(* Logix 5000 project; controller DispersionPlc vendor 1 type 14 code 108 rev 34.11; software revision 34.01; part 17 of 22 *)
(* tags used below, declared in another part *)
   _JISdebug : DINT;
   AFI : BOOL;
   AG4302_LLP_Alarm : BOOL;
   Current4302FQ : REAL;
   DPT_4302_Holding : REAL;
   Estop_Disp : ALIAS FOR Local:3:I.Data.1;
   FIT_4302_1 : AStd_AnalogInput;
   FIT_4305_xx : AStd_AnalogInput;
   K400_PhaseTransfer : AStd_PLI;
   LS_4302_High : BOOL;
   PIC_4302_3 : AStd_PIDInterface;
   RO_HE4305_PhaseROWaterAddition : AStd_PLI;
   SPARE_I402 : ALIAS FOR Local:4:I.Data.2;
   SPARE_I403 : ALIAS FOR Local:4:I.Data.3;
   SPARE_I408 : ALIAS FOR Local:4:I.Data.8;
   SPARE_I409 : ALIAS FOR Local:4:I.Data.9;
   SPARE_O512 : ALIAS FOR Local:5:O.Data.12;
   SPARE_O513 : ALIAS FOR Local:5:O.Data.13;
   SPARE_O605 : ALIAS FOR Local:6:O.Data.5;
   TIT_4305_1 : AStd_AnalogInput;
   V4306_PhaseTransfer : AStd_PLI;
   V4307_PhaseTransfer : AStd_PLI;
   VFD_4302_1 : AStd_VFD;
   VFD_P_4302_2 : AStd_VFD;
   WIT_4302_1 : AStd_AnalogInput;
   WIT_4302_1_AOI : AStd_AI_AOI;
   XV_4301_8 : AStd_VlvOC;
   XV_4302_10 : AStd_VlvOC;
   XV_4302_10_AOI : AStd_VlvOC_AOI;
   XV_4302_10_IOpn : BOOL;
   XV_4302_10_OCls : BOOL;
   XV_4302_12 : AStd_VlvOC;
   XV_4302_12_AOI : AStd_VlvOC_AOI;
   XV_4302_12_OCls : BOOL;
   XV_4302_13 : AStd_VlvOC;
   XV_4302_13_AOI : AStd_VlvOC_AOI;
   XV_4302_13_ClosedI : ALIAS FOR Local:1:I.Data[27].23;
   XV_4302_13_OCls : BOOL;
   XV_4302_13_OpenC : ALIAS FOR Local:1:O.Data[12].17;
   XV_4302_13_OpenI : ALIAS FOR Local:1:I.Data[27].24;
   XV_4302_2 : AStd_VlvOC;
   XV_4302_2_AOI : AStd_VlvOC_AOI;
   XV_4302_2_ICls : BOOL;
   XV_4302_2_IOpn : BOOL;
   XV_4302_2_OCls : BOOL;
   XV_4302_2_OOpn : BOOL;
   XV_4302_3 : AStd_VlvOC;
   XV_4302_3_AOI : AStd_VlvOC_AOI;
   XV_4302_3_ICls : BOOL;
   XV_4302_3_IOpn : BOOL;
   XV_4302_3_OCls : BOOL;
   XV_4302_3_OOpn : BOOL;
   XV_4302_4 : AStd_VlvOC;
   XV_4302_4_AOI : AStd_VlvOC_AOI;
   XV_4302_4_ICls : BOOL;
   XV_4302_4_IOpn : BOOL;
   XV_4302_4_OCls : BOOL;
   XV_4302_4_OOpn : BOOL;
   XV_4302_5 : AStd_VlvOC;
   XV_4302_5_AOI : AStd_VlvOC_AOI;
   XV_4302_5_IOpn : BOOL;
   XV_4302_5_OCls : BOOL;
   XV_4302_6 : AStd_VlvOC;
   XV_4302_6_AOI : AStd_VlvOC_AOI;
   XV_4302_6_IOpn : BOOL;
   XV_4302_6_OCls : BOOL;
   XV_4302_7 : AStd_VlvOC;
   XV_4302_7_AOI : AStd_VlvOC_AOI;
   XV_4302_7_IOpn : BOOL;
   XV_4302_7_OCls : BOOL;
   XV_4302_8 : AStd_VlvOC;
   XV_4302_8_AOI : AStd_VlvOC_AOI;
   XV_4302_8_IOpn : BOOL;
   XV_4302_8_OCls : BOOL;
   XV_4302_9 : AStd_VlvOC;
   XV_4306_3 : AStd_VlvOC;
   XV_4306_5 : AStd_VlvOC;
   XV_4307_3 : AStd_VlvOC;
   XV_4307_6 : AStd_VlvOC;
   XV_S52_2 : AStd_VlvOC;
(* Unit_T4302, continued *)

ROUTINE Device_WIT_4302_1   (* ladder *)
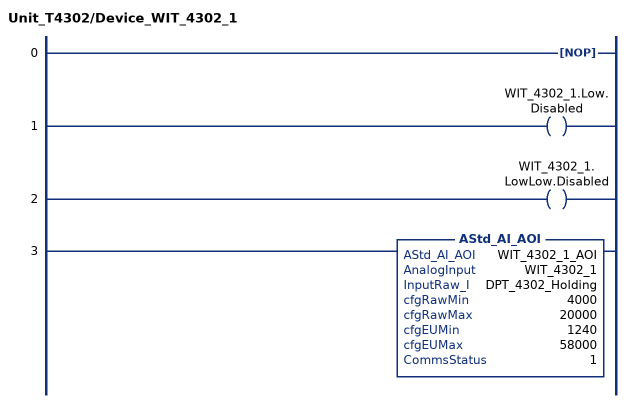
   0: NOP();
   1: OTE(WIT_4302_1.Low.Disabled);
   2: OTE(WIT_4302_1.LowLow.Disabled);
   3: AStd_AI_AOI(WIT_4302_1_AOI,WIT_4302_1,DPT_4302_Holding,4000,20000,1240,58000,1);
END_ROUTINE

ROUTINE Device_XV_4302_10   (* ladder *)
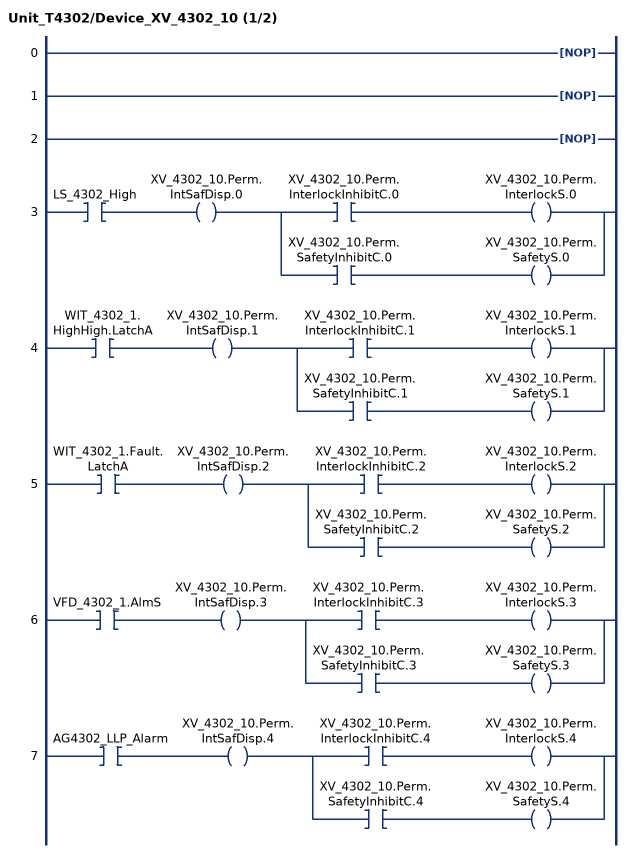
   0: NOP();
   1: NOP();
   2: NOP();
   3: XIC(LS_4302_High)OTE(XV_4302_10.Perm.IntSafDisp.0)[XIC(XV_4302_10.Perm.InterlockInhibitC.0) OTE(XV_4302_10.Perm.InterlockS.0) ,XIC(XV_4302_10.Perm.SafetyInhibitC.0) OTE(XV_4302_10.Perm.SafetyS.0) ];
   4: XIC(WIT_4302_1.HighHigh.LatchA)OTE(XV_4302_10.Perm.IntSafDisp.1)[XIC(XV_4302_10.Perm.InterlockInhibitC.1) OTE(XV_4302_10.Perm.InterlockS.1) ,XIC(XV_4302_10.Perm.SafetyInhibitC.1) OTE(XV_4302_10.Perm.SafetyS.1) ];
   5: XIC(WIT_4302_1.Fault.LatchA)OTE(XV_4302_10.Perm.IntSafDisp.2)[XIC(XV_4302_10.Perm.InterlockInhibitC.2) OTE(XV_4302_10.Perm.InterlockS.2) ,XIC(XV_4302_10.Perm.SafetyInhibitC.2) OTE(XV_4302_10.Perm.SafetyS.2) ];
   6: XIC(VFD_4302_1.AlmS)OTE(XV_4302_10.Perm.IntSafDisp.3)[XIC(XV_4302_10.Perm.InterlockInhibitC.3) OTE(XV_4302_10.Perm.InterlockS.3) ,XIC(XV_4302_10.Perm.SafetyInhibitC.3) OTE(XV_4302_10.Perm.SafetyS.3) ];
   7: XIC(AG4302_LLP_Alarm)OTE(XV_4302_10.Perm.IntSafDisp.4)[XIC(XV_4302_10.Perm.InterlockInhibitC.4) OTE(XV_4302_10.Perm.InterlockS.4) ,XIC(XV_4302_10.Perm.SafetyInhibitC.4) OTE(XV_4302_10.Perm.SafetyS.4) ];
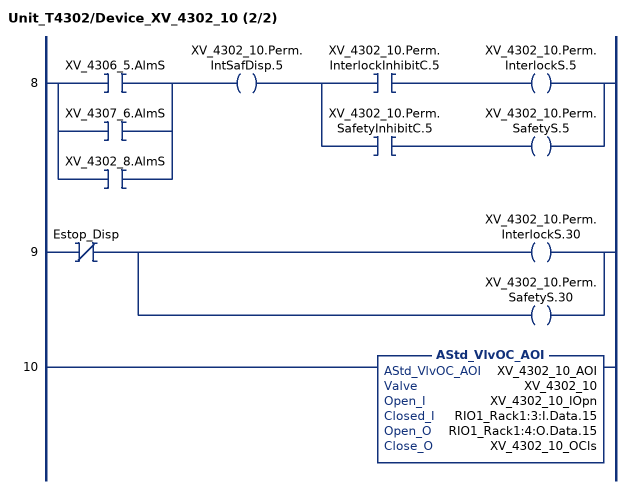
   8: [XIC(XV_4306_5.AlmS) ,XIC(XV_4307_6.AlmS) ,XIC(XV_4302_8.AlmS) ]OTE(XV_4302_10.Perm.IntSafDisp.5)[XIC(XV_4302_10.Perm.InterlockInhibitC.5) OTE(XV_4302_10.Perm.InterlockS.5) ,XIC(XV_4302_10.Perm.SafetyInhibitC.5) OTE(XV_4302_10.Perm.SafetyS.5) ];
   9: XIO(Estop_Disp)[OTE(XV_4302_10.Perm.InterlockS.30) ,OTE(XV_4302_10.Perm.SafetyS.30) ];
   10: AStd_VlvOC_AOI(XV_4302_10_AOI,XV_4302_10,XV_4302_10_IOpn,RIO1_Rack1:3:I.Data.15,RIO1_Rack1:4:O.Data.15,XV_4302_10_OCls);
END_ROUTINE

ROUTINE Device_XV_4302_12   (* ladder *)
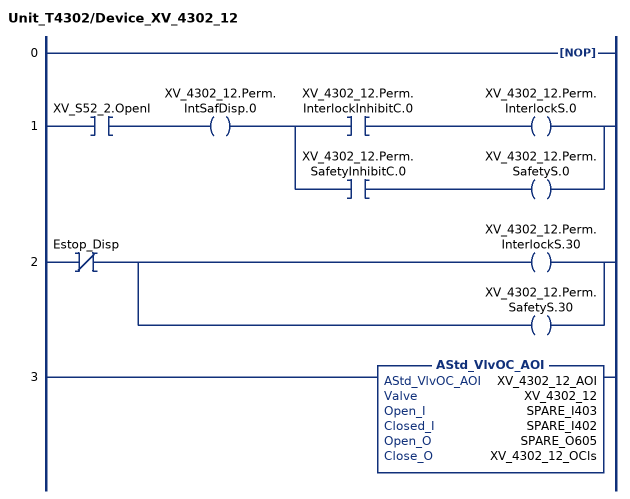
   0: NOP();
   1: XIC(XV_S52_2.OpenI)OTE(XV_4302_12.Perm.IntSafDisp.0)[XIC(XV_4302_12.Perm.InterlockInhibitC.0) OTE(XV_4302_12.Perm.InterlockS.0) ,XIC(XV_4302_12.Perm.SafetyInhibitC.0) OTE(XV_4302_12.Perm.SafetyS.0) ];
   2: XIO(Estop_Disp)[OTE(XV_4302_12.Perm.InterlockS.30) ,OTE(XV_4302_12.Perm.SafetyS.30) ];
   3: AStd_VlvOC_AOI(XV_4302_12_AOI,XV_4302_12,SPARE_I403,SPARE_I402,SPARE_O605,XV_4302_12_OCls);
END_ROUTINE

ROUTINE Device_XV_4302_13   (* ladder *)
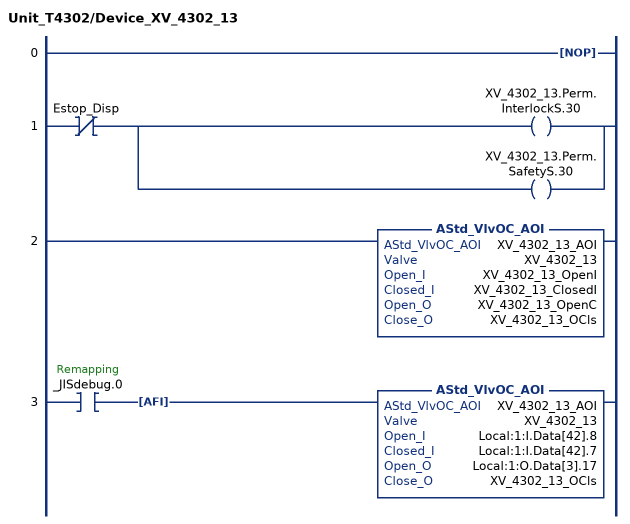
   0: NOP();
   1: XIO(Estop_Disp)[OTE(XV_4302_13.Perm.InterlockS.30) ,OTE(XV_4302_13.Perm.SafetyS.30) ];
   2: AStd_VlvOC_AOI(XV_4302_13_AOI,XV_4302_13,XV_4302_13_OpenI,XV_4302_13_ClosedI,XV_4302_13_OpenC,XV_4302_13_OCls);
   3: XIC(_JISdebug.0)AFI()AStd_VlvOC_AOI(XV_4302_13_AOI,XV_4302_13,Local:1:I.Data[42].8,Local:1:I.Data[42].7,Local:1:O.Data[3].17,XV_4302_13_OCls);
END_ROUTINE

ROUTINE Device_XV_4302_2   (* ladder *)
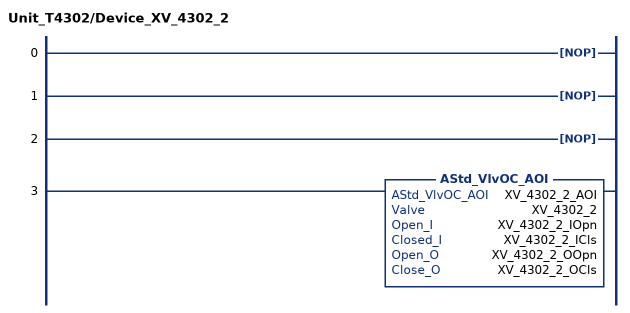
   0: NOP();
   1: NOP();
   2: NOP();
   3: AStd_VlvOC_AOI(XV_4302_2_AOI,XV_4302_2,XV_4302_2_IOpn,XV_4302_2_ICls,XV_4302_2_OOpn,XV_4302_2_OCls);
END_ROUTINE

ROUTINE Device_XV_4302_3   (* ladder *)
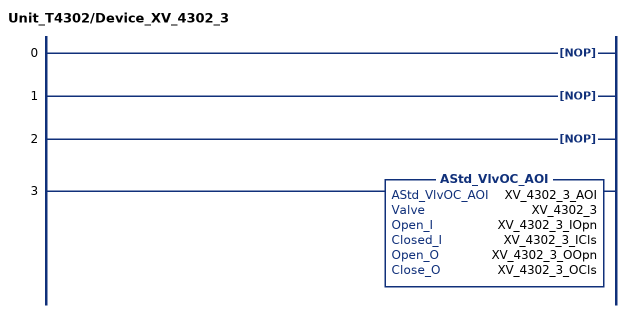
   0: NOP();
   1: NOP();
   2: NOP();
   3: AStd_VlvOC_AOI(XV_4302_3_AOI,XV_4302_3,XV_4302_3_IOpn,XV_4302_3_ICls,XV_4302_3_OOpn,XV_4302_3_OCls);
END_ROUTINE

ROUTINE Device_XV_4302_4   (* ladder *)
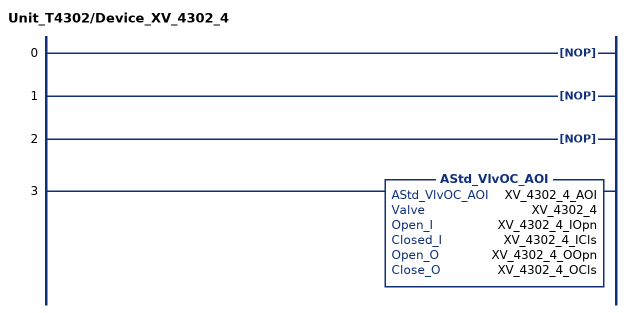
   0: NOP();
   1: NOP();
   2: NOP();
   3: AStd_VlvOC_AOI(XV_4302_4_AOI,XV_4302_4,XV_4302_4_IOpn,XV_4302_4_ICls,XV_4302_4_OOpn,XV_4302_4_OCls);
END_ROUTINE

ROUTINE Device_XV_4302_5   (* ladder *)
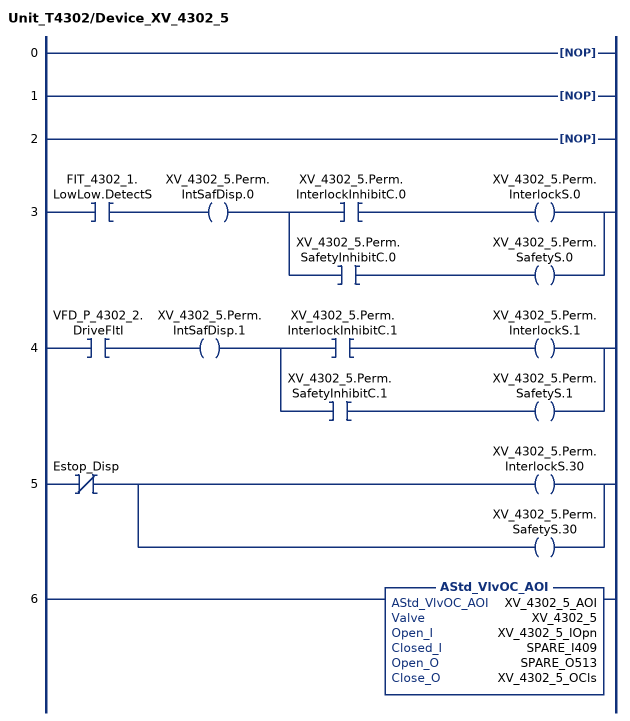
   0: NOP();
   1: NOP();
   2: NOP();
   3: XIC(FIT_4302_1.LowLow.DetectS)OTE(XV_4302_5.Perm.IntSafDisp.0)[XIC(XV_4302_5.Perm.InterlockInhibitC.0) OTE(XV_4302_5.Perm.InterlockS.0) ,XIC(XV_4302_5.Perm.SafetyInhibitC.0) OTE(XV_4302_5.Perm.SafetyS.0) ];
   4: XIC(VFD_P_4302_2.DriveFltI)OTE(XV_4302_5.Perm.IntSafDisp.1)[XIC(XV_4302_5.Perm.InterlockInhibitC.1) OTE(XV_4302_5.Perm.InterlockS.1) ,XIC(XV_4302_5.Perm.SafetyInhibitC.1) OTE(XV_4302_5.Perm.SafetyS.1) ];
   5: XIO(Estop_Disp)[OTE(XV_4302_5.Perm.InterlockS.30) ,OTE(XV_4302_5.Perm.SafetyS.30) ];
   6: AStd_VlvOC_AOI(XV_4302_5_AOI,XV_4302_5,XV_4302_5_IOpn,SPARE_I409,SPARE_O513,XV_4302_5_OCls);
END_ROUTINE

ROUTINE Device_XV_4302_6   (* ladder *)
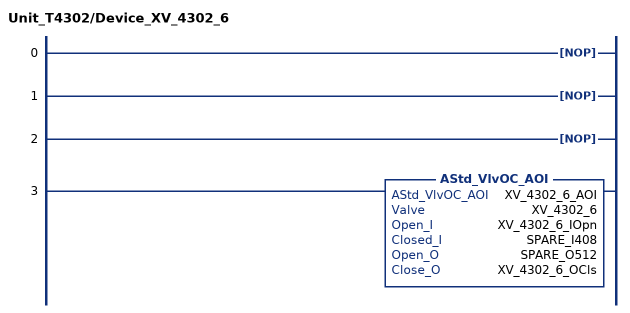
   0: NOP();
   1: NOP();
   2: NOP();
   3: AStd_VlvOC_AOI(XV_4302_6_AOI,XV_4302_6,XV_4302_6_IOpn,SPARE_I408,SPARE_O512,XV_4302_6_OCls);
END_ROUTINE

ROUTINE Device_XV_4302_7   (* ladder *)
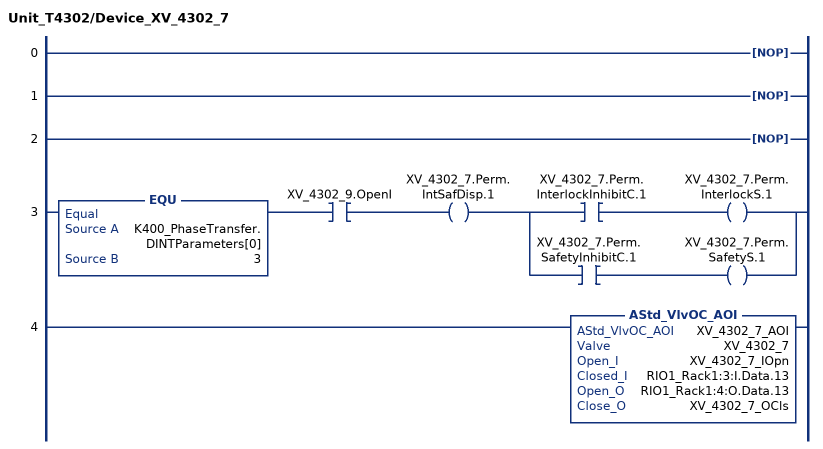
   0: NOP();
   1: NOP();
   2: NOP();
   3: EQU(K400_PhaseTransfer.DINTParameters[0],3)XIC(XV_4302_9.OpenI)OTE(XV_4302_7.Perm.IntSafDisp.1)[XIC(XV_4302_7.Perm.InterlockInhibitC.1) OTE(XV_4302_7.Perm.InterlockS.1) ,XIC(XV_4302_7.Perm.SafetyInhibitC.1) OTE(XV_4302_7.Perm.SafetyS.1) ];
   4: AStd_VlvOC_AOI(XV_4302_7_AOI,XV_4302_7,XV_4302_7_IOpn,RIO1_Rack1:3:I.Data.13,RIO1_Rack1:4:O.Data.13,XV_4302_7_OCls);
END_ROUTINE

ROUTINE Device_XV_4302_8   (* ladder *)
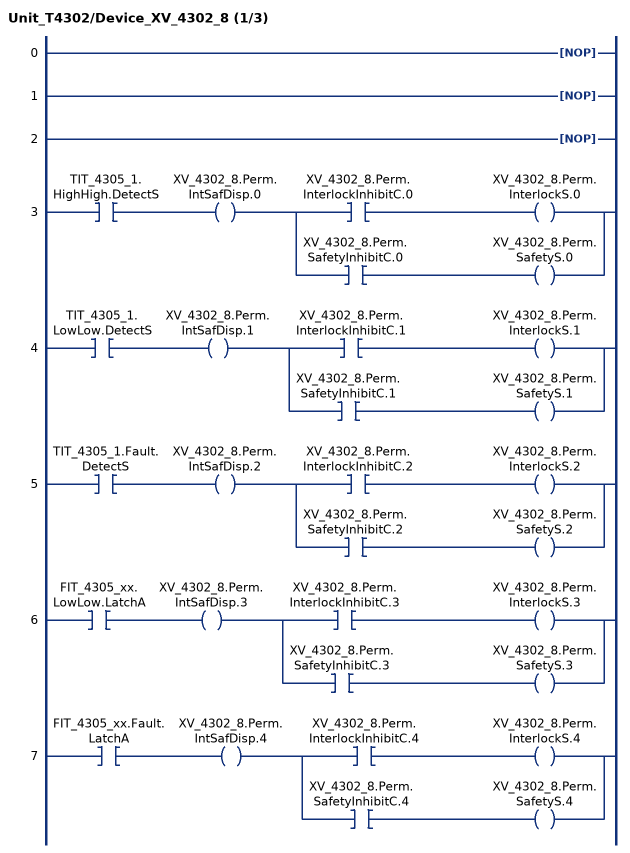
   0: NOP();
   1: NOP();
   2: NOP();
   3: XIC(TIT_4305_1.HighHigh.DetectS)OTE(XV_4302_8.Perm.IntSafDisp.0)[XIC(XV_4302_8.Perm.InterlockInhibitC.0) OTE(XV_4302_8.Perm.InterlockS.0) ,XIC(XV_4302_8.Perm.SafetyInhibitC.0) OTE(XV_4302_8.Perm.SafetyS.0) ];
   4: XIC(TIT_4305_1.LowLow.DetectS)OTE(XV_4302_8.Perm.IntSafDisp.1)[XIC(XV_4302_8.Perm.InterlockInhibitC.1) OTE(XV_4302_8.Perm.InterlockS.1) ,XIC(XV_4302_8.Perm.SafetyInhibitC.1) OTE(XV_4302_8.Perm.SafetyS.1) ];
   5: XIC(TIT_4305_1.Fault.DetectS)OTE(XV_4302_8.Perm.IntSafDisp.2)[XIC(XV_4302_8.Perm.InterlockInhibitC.2) OTE(XV_4302_8.Perm.InterlockS.2) ,XIC(XV_4302_8.Perm.SafetyInhibitC.2) OTE(XV_4302_8.Perm.SafetyS.2) ];
   6: XIC(FIT_4305_xx.LowLow.LatchA)OTE(XV_4302_8.Perm.IntSafDisp.3)[XIC(XV_4302_8.Perm.InterlockInhibitC.3) OTE(XV_4302_8.Perm.InterlockS.3) ,XIC(XV_4302_8.Perm.SafetyInhibitC.3) OTE(XV_4302_8.Perm.SafetyS.3) ];
   7: XIC(FIT_4305_xx.Fault.LatchA)OTE(XV_4302_8.Perm.IntSafDisp.4)[XIC(XV_4302_8.Perm.InterlockInhibitC.4) OTE(XV_4302_8.Perm.InterlockS.4) ,XIC(XV_4302_8.Perm.SafetyInhibitC.4) OTE(XV_4302_8.Perm.SafetyS.4) ];
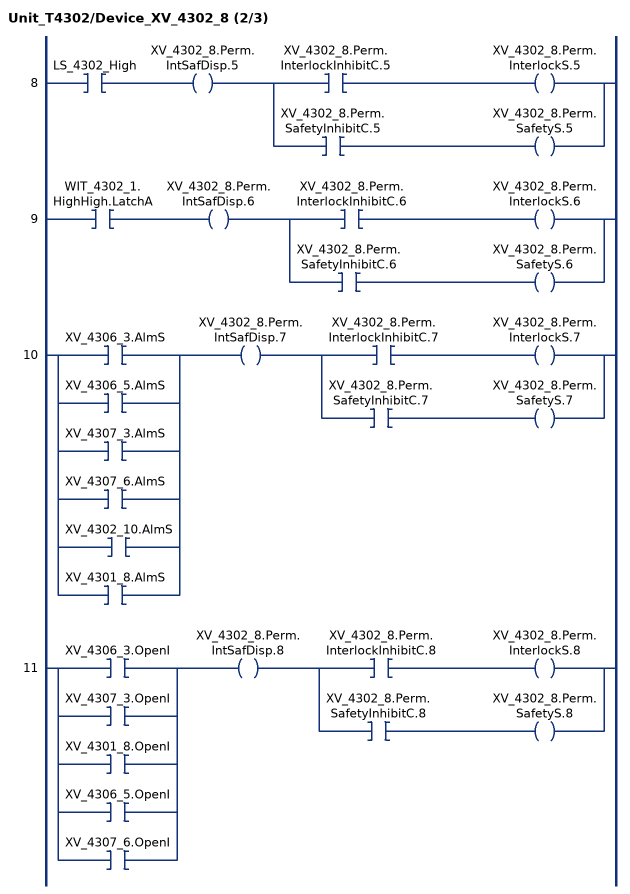
   8: XIC(LS_4302_High)OTE(XV_4302_8.Perm.IntSafDisp.5)[XIC(XV_4302_8.Perm.InterlockInhibitC.5) OTE(XV_4302_8.Perm.InterlockS.5) ,XIC(XV_4302_8.Perm.SafetyInhibitC.5) OTE(XV_4302_8.Perm.SafetyS.5) ];
   9: XIC(WIT_4302_1.HighHigh.LatchA)OTE(XV_4302_8.Perm.IntSafDisp.6)[XIC(XV_4302_8.Perm.InterlockInhibitC.6) OTE(XV_4302_8.Perm.InterlockS.6) ,XIC(XV_4302_8.Perm.SafetyInhibitC.6) OTE(XV_4302_8.Perm.SafetyS.6) ];
   10: [XIC(XV_4306_3.AlmS) ,XIC(XV_4306_5.AlmS) ,XIC(XV_4307_3.AlmS) ,XIC(XV_4307_6.AlmS) ,XIC(XV_4302_10.AlmS) ,XIC(XV_4301_8.AlmS) ]OTE(XV_4302_8.Perm.IntSafDisp.7)[XIC(XV_4302_8.Perm.InterlockInhibitC.7) OTE(XV_4302_8.Perm.InterlockS.7) ,XIC(XV_4302_8.Perm.SafetyInhibitC.7) OTE(XV_4302_8.Perm.SafetyS.7) ];
   11: [XIC(XV_4306_3.OpenI) ,XIC(XV_4307_3.OpenI) ,XIC(XV_4301_8.OpenI) ,XIC(XV_4306_5.OpenI) ,XIC(XV_4307_6.OpenI) ]OTE(XV_4302_8.Perm.IntSafDisp.8)[XIC(XV_4302_8.Perm.InterlockInhibitC.8) OTE(XV_4302_8.Perm.InterlockS.8) ,XIC(XV_4302_8.Perm.SafetyInhibitC.8) OTE(XV_4302_8.Perm.SafetyS.8) ];
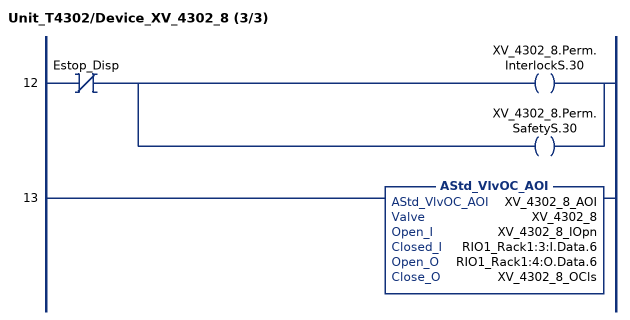
   12: XIO(Estop_Disp)[OTE(XV_4302_8.Perm.InterlockS.30) ,OTE(XV_4302_8.Perm.SafetyS.30) ];
   13: AStd_VlvOC_AOI(XV_4302_8_AOI,XV_4302_8,XV_4302_8_IOpn,RIO1_Rack1:3:I.Data.6,RIO1_Rack1:4:O.Data.6,XV_4302_8_OCls);
END_ROUTINE

ROUTINE FQ_4302_2   (* ladder *)
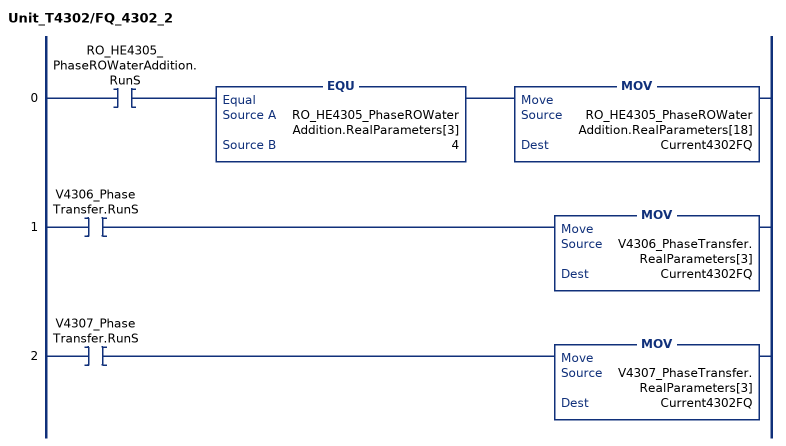
   0: XIC(RO_HE4305_PhaseROWaterAddition.RunS)EQU(RO_HE4305_PhaseROWaterAddition.RealParameters[3],4)MOV(RO_HE4305_PhaseROWaterAddition.RealParameters[18],Current4302FQ);
   1: XIC(V4306_PhaseTransfer.RunS)MOV(V4306_PhaseTransfer.RealParameters[3],Current4302FQ);
   2: XIC(V4307_PhaseTransfer.RunS)MOV(V4307_PhaseTransfer.RealParameters[3],Current4302FQ);
END_ROUTINE

ROUTINE MainRoutine   (* ladder *)
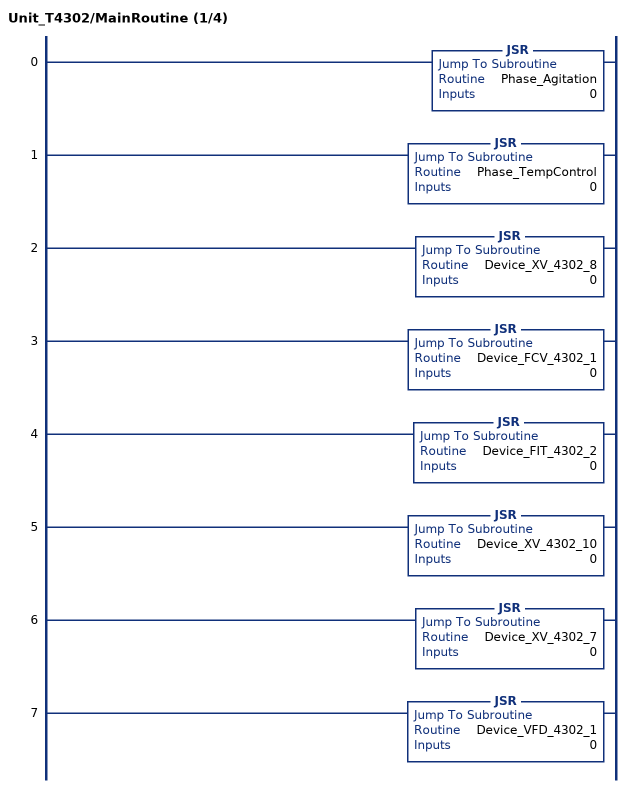
   0: JSR(Phase_Agitation,0);
   1: JSR(Phase_TempControl,0);
   2: JSR(Device_XV_4302_8,0);
   3: JSR(Device_FCV_4302_1,0);
   4: JSR(Device_FIT_4302_2,0);
   5: JSR(Device_XV_4302_10,0);
   6: JSR(Device_XV_4302_7,0);
   7: JSR(Device_VFD_4302_1,0);
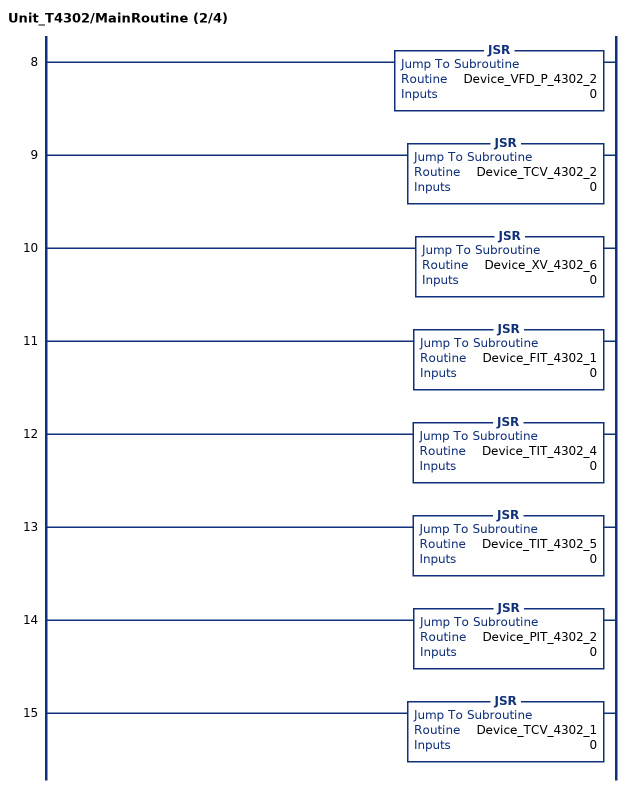
   8: JSR(Device_VFD_P_4302_2,0);
   9: JSR(Device_TCV_4302_2,0);
   10: JSR(Device_XV_4302_6,0);
   11: JSR(Device_FIT_4302_1,0);
   12: JSR(Device_TIT_4302_4,0);
   13: JSR(Device_TIT_4302_5,0);
   14: JSR(Device_PIT_4302_2,0);
   15: JSR(Device_TCV_4302_1,0);
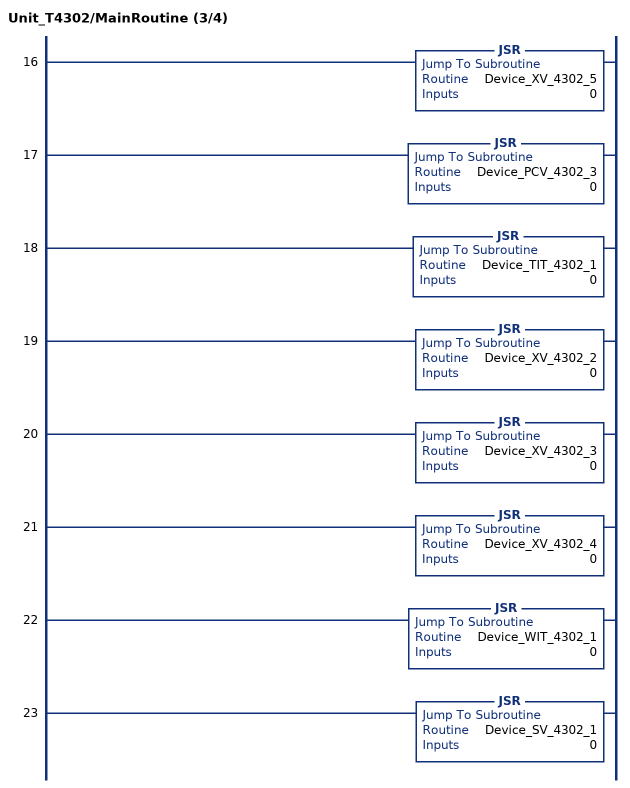
   16: JSR(Device_XV_4302_5,0);
   17: JSR(Device_PCV_4302_3,0);
   18: JSR(Device_TIT_4302_1,0);
   19: JSR(Device_XV_4302_2,0);
   20: JSR(Device_XV_4302_3,0);
   21: JSR(Device_XV_4302_4,0);
   22: JSR(Device_WIT_4302_1,0);
   23: JSR(Device_SV_4302_1,0);
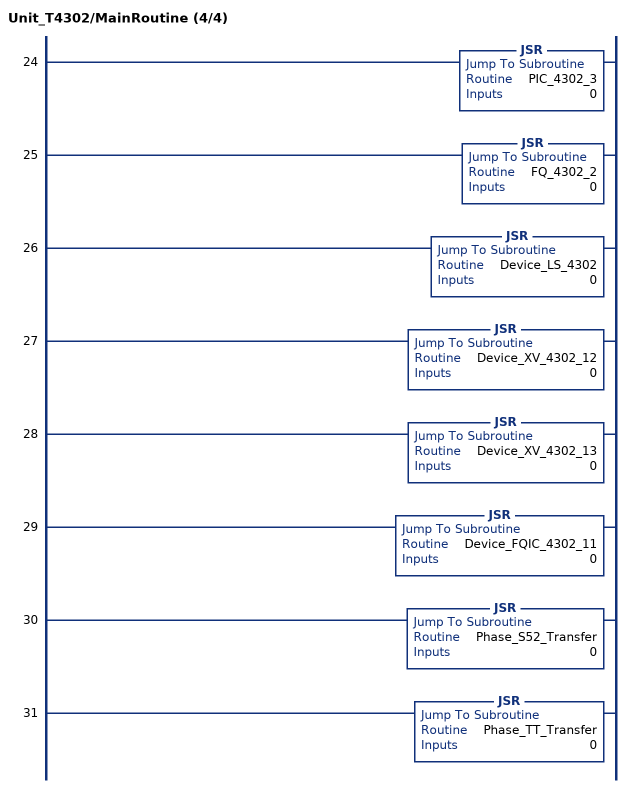
   24: JSR(PIC_4302_3,0);
   25: JSR(FQ_4302_2,0);
   26: JSR(Device_LS_4302,0);
   27: JSR(Device_XV_4302_12,0);
   28: JSR(Device_XV_4302_13,0);
   29: JSR(Device_FQIC_4302_11,0);
   30: JSR(Phase_S52_Transfer,0);
   31: JSR(Phase_TT_Transfer,0);
END_ROUTINE
